(*udt (user defined type) of Beckhoff EP2028-0002 - 8 Point IP67 Rated Digital Output Box:
	auth. Brent Lekx-Toniolo of Toniolo Research & Development Inc.; 
	July 2010; version 1.0*)


TYPE udt_EP2028_002 :
STRUCT
	Q0: BOOL;
	Q1: BOOL;
	Q2: BOOL;
	Q3: BOOL;
	Q4: BOOL;
	Q5: BOOL;
	Q6: BOOL;
	Q7: BOOL;
END_STRUCT
END_TYPE

(* stored: Version 1.1.0.1, ProductVersion 3.1.4024.9
   DUT udt_EP2028_002: Id {e36a88fd-9b59-4296-9bad-2452d6312e87} *)
